(* PLC project TestSuite.project, CODESYS CODESYS V3.5 SP21 Patch 2 *)
(* stored: creationDateTime 2025-09-07T16:10:53.1946689, modificationDateTime 2025-09-07T15:30:20.0228435 *)

PROGRAM PRG_TestRunner
  VAR
    T : FB_Test_ClampF;
  END_VAR

                  T(); // richiama una volta a ciclo
// controlla T.Failures in watch. 0 = OK.
                
END_PROGRAM

FUNCTION_BLOCK FB_Test_ClampF
  VAR
    Failures : UDINT;
    Done : BOOL;
    _ok : BOOL;
  END_VAR

                  // ciclo unico: esegui asserzioni una volta
IF NOT Done THEN
    ExpectTrue(ABS(ClampF(5.0, 0.0, 10.0) - 5.0) < 1e-6, '5 in [0,10]');
    ExpectTrue(ABS(ClampF(-2.0,0.0, 10.0) - 0.0) < 1e-6, '-2 -> 0');
    ExpectTrue(ABS(ClampF(99.0,0.0, 10.0) - 10.0) < 1e-6, '99 -> 10');
    ExpectTrue(ABS(ClampF(0.0, 0.0, 10.0) - 0.0) < 1e-6, 'bordo lo');
    ExpectTrue(ABS(ClampF(10.0,0.0, 10.0) -10.0) < 1e-6, 'bordo hi');
    Done := TRUE;
END_IF
                

METHOD ExpectTrue
  VAR_INPUT
    cond : BOOL;
    msg : STRING;
  END_VAR
                        IF NOT cond THEN
    Failures := Failures + 1;
END_IF
                      
END_METHOD
END_FUNCTION_BLOCK

FUNCTION ClampF : REAL
  VAR_INPUT
    x : REAL;
    lo : REAL;
    hi : REAL;
  END_VAR

                  IF x < lo THEN
    ClampF := lo;
ELSIF x > hi THEN
    ClampF := hi;
ELSE
    ClampF := x;
END_IF
                
END_FUNCTION

CONFIGURATION Application
  RESOURCE Application ON PLC
    TASK Task_test(INTERVAL := T#20ms, PRIORITY := 1);
    PROGRAM PRG_TestRunner WITH Task_test : PRG_TestRunner;
  END_RESOURCE
END_CONFIGURATION
